TYPE T_Enum : E_Enum; END_TYPE

(* stored: Version 1.1.0.1
   DUT T_Enum: Id {cdca9a92-3731-4511-abf0-87964f650eb1} *)
